% RSLogix 500 project I2A-JOB 8-MITCH_BAK019.RSS, saved by version 10.00.00.00 %
PROJECT "ML01B"    % processor: Bul.1763 MicroLogix 1100 Series B %

PROGRAM FILES
  LAD 2   5 rungs

DATA FILES
  O0 OUTPUT  4 elements
  I1 INPUT  6 elements
  S2 STATUS  66 elements
  B3 BINARY  1 elements
  T4 TIMER  1 elements
  C5 COUNTER  1 elements
  R6 CONTROL  1 elements
  N7 INTEGER  1 elements
  F8 FLOAT  1 elements

LADDER 2
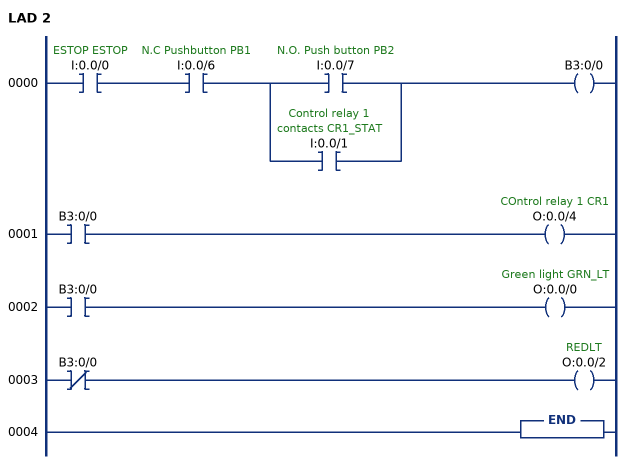
% Rung: 0 %
SOR XIC I:0.0/0 XIC I:0.0/6 BST XIC I:0.0/7 NXB XIC I:0.0/1 BND OTE B3:0/0 EOR
%   I:0.0/0  ESTOP  "ESTOP" %
%   I:0.0/6  PB1  "N.C Pushbutton" %
%   I:0.0/7  PB2  "N.O. Push button" %
%   I:0.0/1  CR1_STAT  "Control relay 1 contacts" %
% Rung: 1 %
SOR XIC B3:0/0 OTE O:0.0/4 EOR
%   O:0.0/4  CR1  "COntrol relay 1" %
% Rung: 2 %
SOR XIC B3:0/0 OTE O:0.0/0 EOR
%   O:0.0/0  GRN_LT  "Green light" %
% Rung: 3 %
SOR XIO B3:0/0 OTE O:0.0/2 EOR
%   O:0.0/2  REDLT %
% Rung: 4 %
SOR END EOR

OTHER DOCUMENTED ADDRESSES
  I:0.0/2  CR2_STAT  "Control relay 2 contacts"
  I:0.0/3  3PSSA  "thre position switch A"
  I:0.0/4  3PSS_B  "Three posision selector switch B"
  I:0.0/5  2PSSA  "2 position selector switch A"
  I:0.0/8  PB3  "N.O pushbutton"
  O:0.0/1  YELLOWLT
  O:0.0/3  BLUELT  "TOM BRADY IS THE GREATEST OF ALL TIME"
  O:0.0/5  CR2  "Control relay 2"
